(* IEC 61131-3 sources: CodesysTest/alpha/export/FBs/FB_FaultHandler.pou, 1 file *)

(* ---- FB_FaultHandler.pou.st ---- *)
(*#-#-#-#-#-#-#-#-#-#---Declaration---#-#-#-#-#-#-#-#-#-#-#-#-#*)

FUNCTION_BLOCK FB_FaultHandler
VAR_INPUT
END_VAR
VAR_OUTPUT
END_VAR
VAR
    faultSourceList : ARRAY[0..100] OF IFault;
    sourcesInList : INT;
END_VAR
(*#-#-#-#-#-#-#-#-#-#---Implementation---#-#-#-#-#-#-#-#-#-#-#-#-#*)
